// Public command interface for a Worker.
INTERFACE I_Worker EXTENDS _I_Worker

// Starts idle job; returns Ok attached, None command busy, Error invalid state or job.
METHOD Start : Result
VAR_INPUT
END_VAR
END_METHOD

// Current worker state.
PROPERTY State : JobState
GET
END_GET
END_PROPERTY

// Requests stop; Busy moves to Done and calls JobExit before returning Idle.
METHOD Stop
VAR_INPUT
END_VAR
END_METHOD

END_INTERFACE

(* stored: Version 1.1.0.1
   Itf I_Worker: Id {cf0ee183-0056-4830-bcdb-219351329d42}
   Method Start: Id {c19e8475-caa0-4669-afd8-6d9af8e07fba}
   Property State: Id {2f9f3114-975b-4331-a00b-ffbc0b3559d9}
   Get Get: Id {ec335181-6e97-4eac-a6fd-5f3b403f44f5}
   Method Stop: Id {ac7127aa-39d4-435f-b5d0-74c0f4a14a7e} *)
